INTERFACE I_Sequenz

METHOD M_Reset : BOOL
VAR_INPUT
END_VAR
END_METHOD

METHOD M_Start : BOOL
VAR_INPUT
END_VAR
END_METHOD

METHOD M_Stop : BOOL
VAR_INPUT
END_VAR
END_METHOD

PROPERTY P_Finished : BOOL
GET
END_GET
END_PROPERTY

PROPERTY P_State : INT
GET
END_GET
END_PROPERTY

END_INTERFACE

(* stored: Version 1.1.0.1
   Itf I_Sequenz: Id {28ceae57-4089-44a8-ae28-9022f28b8d95}
   Method M_Reset: Id {f1f5cbc4-ea4f-4e1f-94b4-19b42d581bee}
   Method M_Start: Id {7595f5ae-7473-40a2-b38e-71430a151be1}
   Method M_Stop: Id {3ff0a064-1a84-478c-95ab-766dafd5e58d}
   Property P_Finished: Id {5d7265bd-3769-47df-a5d8-a2727e912dfe}
   Get Get: Id {f6ec5dc3-e29a-46be-94b5-c4717c14f8d4}
   Property P_State: Id {d4f0c874-60ab-44ff-b287-3e5c50ec6755}
   Get Get: Id {8f2f7291-dc2d-4e33-80a7-4abdfeb82956} *)
